(* CoDeSys 2.3.6.0 project: PLC.pro *)
(* Libraries: STANDARD.LIB 5.6.98 12:03:02 *)

(* Task configuration *)
TASK Standard (PRIORITY := 0, INTERVAL := T#400ms);
	MAIN
END_TASK

(* Global variable list: TwinCAT_Configuration *)
(* Generated automatically by TwinCAT - (read only) *)
VAR_CONFIG
	MAIN.myInput AT %IB0 : BYTE;	(*  ~ {LinkedWith:TIID^Gerät 1 (EtherCAT)^Box 2 (EL9800)^Byte 0^Input} *)
	MAIN.myOutput AT %QB0 : BYTE;	(*  ~ {LinkedWith:TIID^Gerät 1 (EtherCAT)^Box 1 (EL9800)^Byte 0^Output} *)
END_VAR

(* POU MAIN, ST *)
PROGRAM MAIN
VAR
	myInput 		AT%I*	:BYTE;
	myOutput	AT%Q*	:BYTE;

END_VAR
myOutput := myInput;
END_PROGRAM
